SUBAPPLICATION Uebung_055_AX (* DigitalInput_I1 auf DigitalOutput_Q1, mit Plug and Socket *)
  (* Standard: 61499-2; Description: Copyright (c) 2026 Meisterschulen am Ostbahnhof This program and the accompanying materials are made available under the terms of the Eclipse Public License 2.0 which is available at https://www.eclipse.org/legal/epl-2.0/ SPDX-License-Identifier: EPL-2.0 *)
  (* Version 1.0, 2026-09-09, Franz Höpfinger, Meisterschulen am Ostbahnhof, initial API and implementation and/or initial documentation *)
  PACKAGE Uebungen;
  IMPORT logiBUS::io::DI::logiBUS_DI::Input_I1;
  IMPORT logiBUS::io::DQ::logiBUS_DO::Output_Q1;
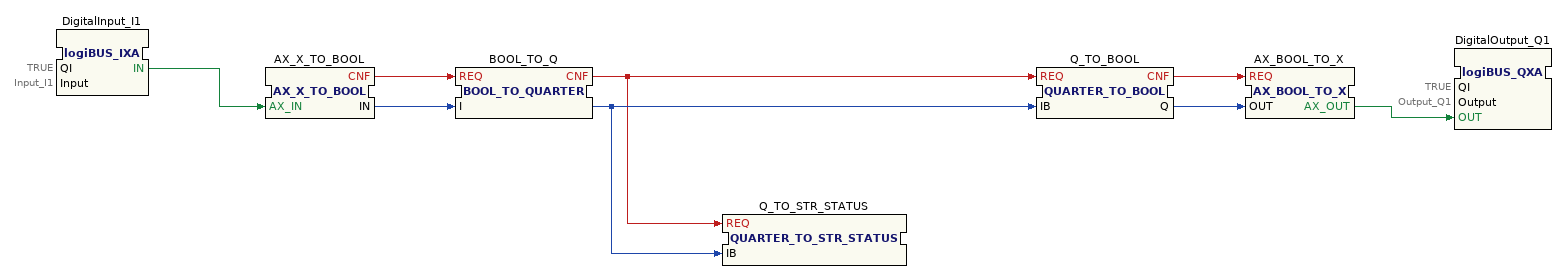
  FBS
    DigitalOutput_Q1 : logiBUS::io::DQ::logiBUS_QXA(QI := TRUE, Output := Output_Q1);
    DigitalInput_I1 : logiBUS::io::DI::logiBUS_IXA(QI := TRUE, Input := Input_I1);
    Q_TO_STR_STATUS : logiBUS::utils::quarter::QUARTER_TO_STR_STATUS;
    Q_TO_BOOL : logiBUS::utils::quarter::QUARTER_TO_BOOL;
    BOOL_TO_Q : logiBUS::utils::quarter::BOOL_TO_QUARTER;
    AX_X_TO_BOOL : adapter::conversion::unidirectional::AX_X_TO_BOOL;
    AX_BOOL_TO_X : adapter::conversion::unidirectional::AX_BOOL_TO_X;
  END_FBS
  EVENT_CONNECTIONS
    Q_TO_BOOL.CNF TO AX_BOOL_TO_X.REQ;
    AX_X_TO_BOOL.CNF TO BOOL_TO_Q.REQ;
    BOOL_TO_Q.CNF TO Q_TO_STR_STATUS.REQ;
    BOOL_TO_Q.CNF TO Q_TO_BOOL.REQ;
  END_CONNECTIONS
  DATA_CONNECTIONS
    Q_TO_BOOL.Q TO AX_BOOL_TO_X.OUT;
    AX_X_TO_BOOL.IN TO BOOL_TO_Q.I;
    BOOL_TO_Q. TO Q_TO_STR_STATUS.IB;
    BOOL_TO_Q. TO Q_TO_BOOL.IB;
  END_CONNECTIONS
  ADAPTER_CONNECTIONS
    DigitalInput_I1.IN TO AX_X_TO_BOOL.AX_IN;
    AX_BOOL_TO_X.AX_OUT TO DigitalOutput_Q1.OUT;
  END_CONNECTIONS
END_SUBAPPLICATION
